(* PLC project Semester-Project-RLW, Unknown RLW-PLC-Command 0.0.1 *)
(* stored: creationDateTime 2024-10-23T22:26:44, modificationDateTime 2024-11-23T23:37:16, version 0.0.1 *)

FUNCTION isWithin5Percent : BOOL
  VAR_INPUT
    In0 : INT;
    In1 : INT;
  END_VAR
  VAR
    RangeHigh : INT;
    RangeLow : INT;
    In0IsLessThanHigh : BOOL;
    In0IsGreaterThanLow : BOOL;
  END_VAR

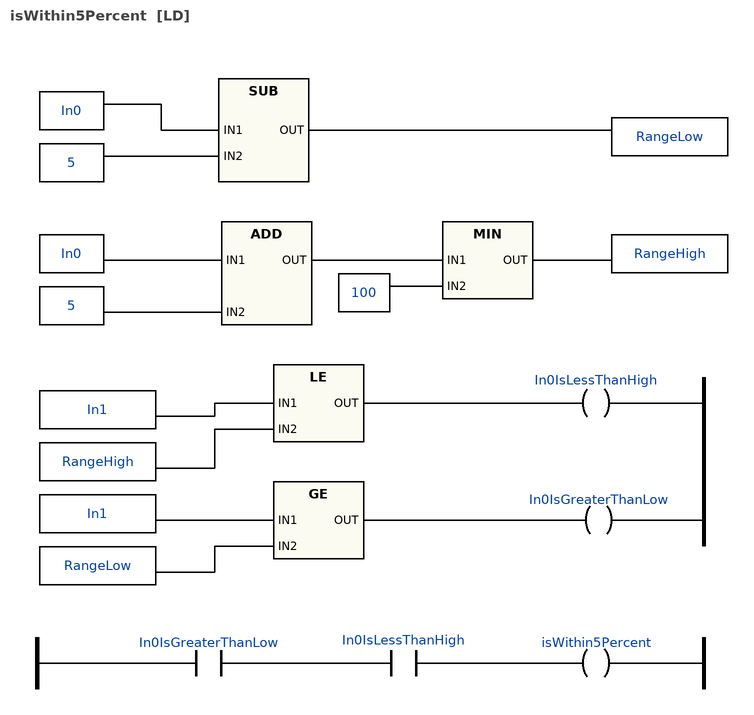
(* LD diagram, written out as Structured Text *)
RangeLow := In0 - 5;
RangeHigh := MIN(In0 + 5, 100);
In0IsLessThanHigh := In1 <= RangeHigh;
In0IsGreaterThanLow := In1 >= RangeLow;
isWithin5Percent := In0IsGreaterThanLow AND In0IsLessThanHigh;
END_FUNCTION

(* Based upon boolean inputs, returns a precentage that the isolation valve should close at. *)
FUNCTION SelectIsolationValveValue : INT
  VAR_INPUT
    SiteAlarmOverride : BOOL;  (* If high, override real num output to 0.0 *)
    BoosterPumpLogicalStatus : BOOL;  (* If high, means booster pump is working and isolation valve output should be 1.0, if low, default to 0.5 *)
  END_VAR

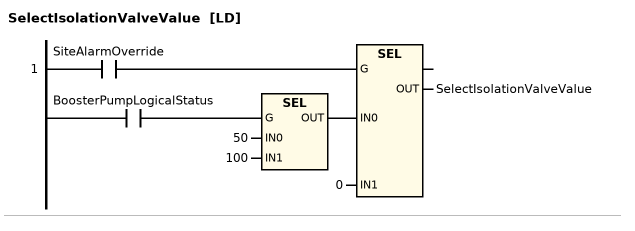
(* LD diagram, written out as Structured Text *)
SelectIsolationValveValue := SEL(SiteAlarmOverride, SEL(BoosterPumpLogicalStatus, 50, 100), 0);
END_FUNCTION

FUNCTION SetFlowSensorAlarm : BOOL
  VAR_INPUT
    IsolationValveStatus : INT;
    FlowRateSensor : INT;
  END_VAR

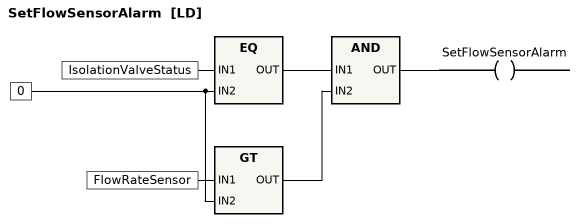
(* LD diagram, written out as Structured Text *)
SetFlowSensorAlarm := IsolationValveStatus = 0 AND FlowRateSensor > 0;
END_FUNCTION

PROGRAM DCSProgramSector
  VAR
    FlowRateSensor0 AT %IW0 : INT := 20;
    FlowRateSensor1 AT %IW1 : INT := 33;
    FlowRateSensor2 AT %IW2 : INT := 46;
    BoosterPumpStatus0 AT %IX0.0 : BOOL := True;
    BoosterPumpStatus1 AT %IX0.1 : BOOL := False;
    BoosterPumpStatus2 AT %IX0.2 : BOOL := False;
    IsolationValveStatus0 AT %IW3 : INT := 50;
    IsolationValveStatus1 AT %IW4 : INT := 50;
    IsolationValveStatus2 AT %IW5 : INT := 50;
    GeneralSiteAlarm0 AT %IX0.3 : BOOL := False;
  END_VAR
  VAR_EXTERNAL
    BoosterPumpCommand0 : BOOL;
    BoosterPumpCommand1 : BOOL;
    BoosterPumpCommand2 : BOOL;
  END_VAR
  VAR
    BoosterPumpAlarm0 AT %QX0.5 : BOOL;
    BoosterPumpAlarm1 AT %QX0.6 : BOOL;
    BoosterPumpAlarm2 AT %QX0.7 : BOOL;
    IsolationValveAlarm0 AT %QX1.0 : BOOL;
    IsolationValveAlarm1 AT %QX1.1 : BOOL;
    IsolationValveAlarm2 AT %QX1.2 : BOOL;
    FlowSensorAlarm0 AT %QX1.3 : BOOL;
    FlowSensorAlarm1 AT %QX1.4 : BOOL;
    FlowSensorAlarm2 AT %QX1.5 : BOOL;
    FlowRateAlarm0 AT %QX4.3 : BOOL;
    FlowRateAlarm1 AT %QX4.4 : BOOL;
    FlowRateAlarm2 AT %QX4.5 : BOOL;
  END_VAR
  VAR_EXTERNAL
    IsolationValveCommand0 : INT;
    IsolationValveCommand1 : INT;
    IsolationValveCommand2 : INT;
  END_VAR
  VAR CONSTANT
    FlowSensorMaxCapacity AT %MW0 : INT := 50;
  END_VAR
  VAR  (* added by the conversion: wires and edge detectors of the diagram *)
    _SelectIsolationValveValue19_OUT : INT;
    _SelectIsolationValveValue25_OUT : INT;
    _SelectIsolationValveValue92_OUT : INT;
  END_VAR

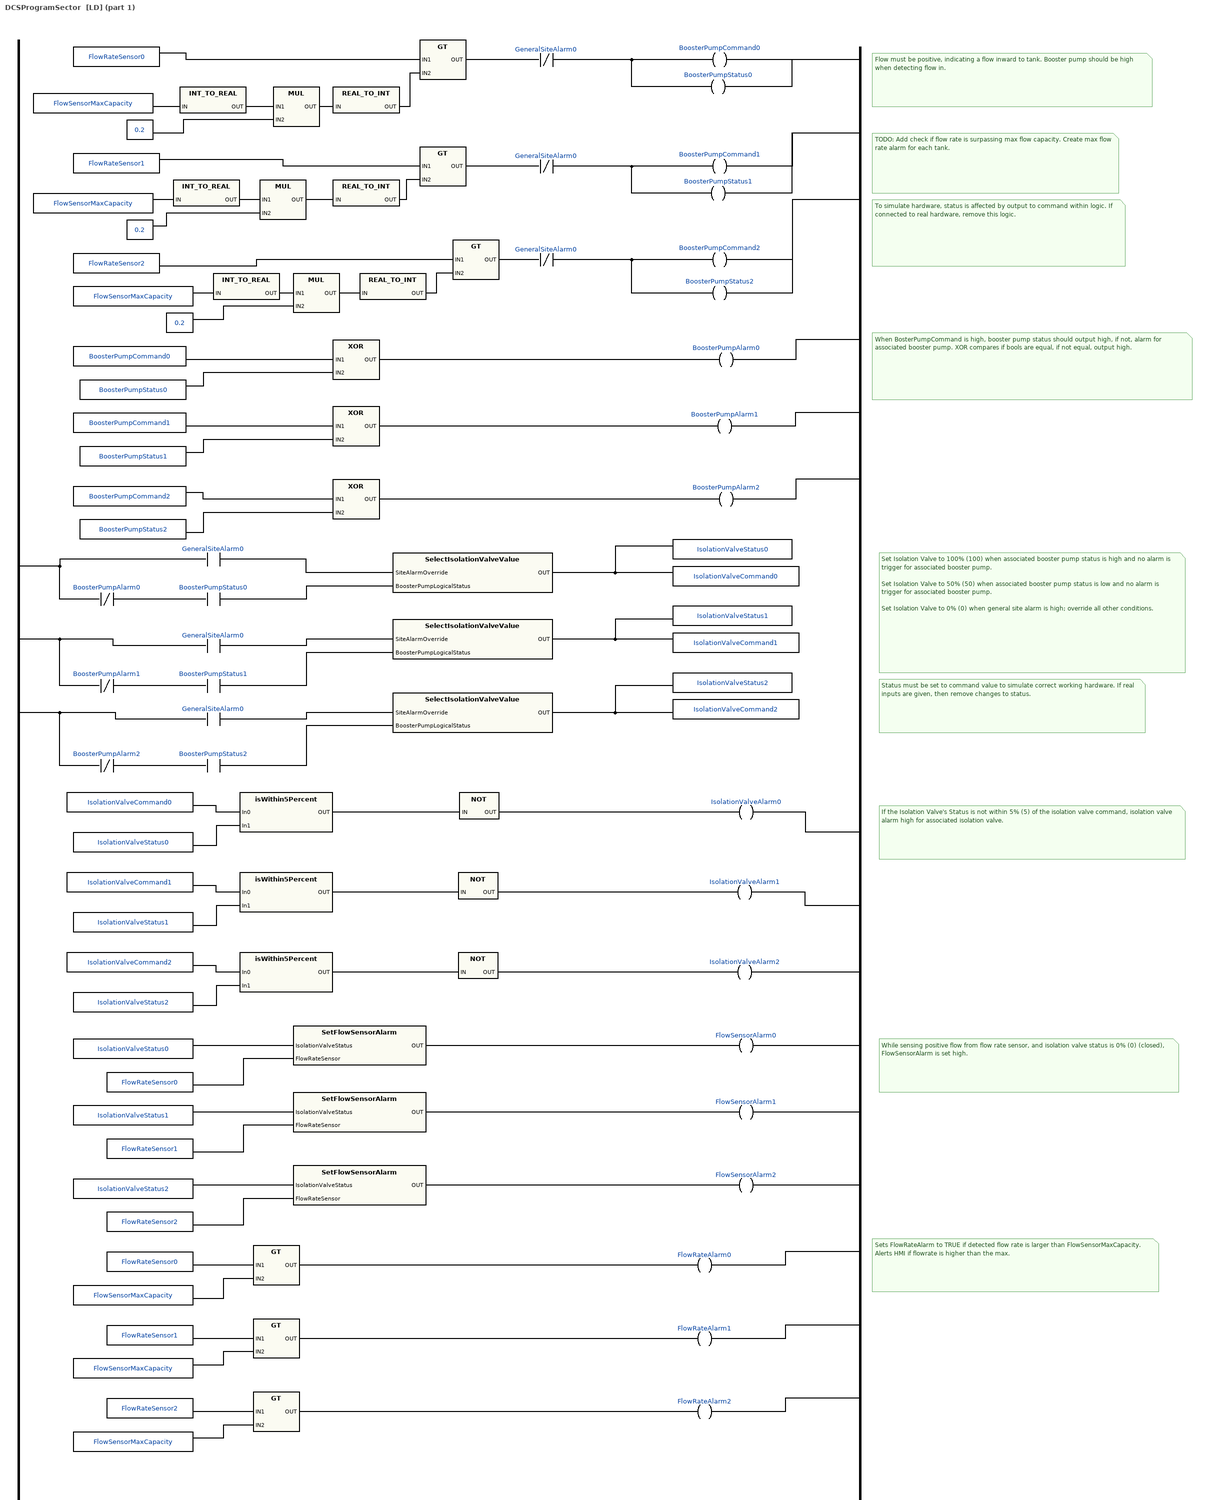
(* LD diagram, written out as Structured Text *)
(* Flow must be positive, indicating a flow inward to tank. Booster pump should be high when detecting flow in. *)
BoosterPumpCommand0 := FlowRateSensor0 > REAL_TO_INT(INT_TO_REAL(FlowSensorMaxCapacity) * 0.2) AND NOT GeneralSiteAlarm0;
(* TODO: Add check if flow rate is surpassing max flow capacity. Create max flow rate alarm for each tank. *)
BoosterPumpCommand1 := FlowRateSensor1 > REAL_TO_INT(INT_TO_REAL(FlowSensorMaxCapacity) * 0.2) AND NOT GeneralSiteAlarm0;
(* To simulate hardware, status is affected by output to command within logic. If connected to real hardware, remove this logic. *)
BoosterPumpCommand2 := FlowRateSensor2 > REAL_TO_INT(INT_TO_REAL(FlowSensorMaxCapacity) * 0.2) AND NOT GeneralSiteAlarm0;
(* When BosterPumpCommand is high, booster pump status should output high, if not, alarm for associated booster pump. XOR compares if bools are equal, if not equal, output high. *)
BoosterPumpAlarm0 := BoosterPumpCommand0 XOR BoosterPumpStatus0;
BoosterPumpAlarm2 := BoosterPumpCommand2 XOR BoosterPumpStatus2;
(* Set Isolation Valve to 100% (100) when associated booster pump status is high and no alarm is trigger for associated booster pump.

Set Isolation Valve to 50% (50) when associated booster pump status is low and no alarm is trigger for associated booster pump.

Set Isolation Valve to 0% (0) when general site alarm is high; override all other conditions. *)
_SelectIsolationValveValue19_OUT := SelectIsolationValveValue(GeneralSiteAlarm0, NOT BoosterPumpAlarm1 AND BoosterPumpStatus1);
IsolationValveCommand1 := _SelectIsolationValveValue19_OUT;
(* Status must be set to command value to simulate correct working hardware. If real inputs are given, then remove changes to status. *)
_SelectIsolationValveValue25_OUT := SelectIsolationValveValue(GeneralSiteAlarm0, NOT BoosterPumpAlarm2 AND BoosterPumpStatus2);
IsolationValveCommand2 := _SelectIsolationValveValue25_OUT;
(* If the Isolation Valve's Status is not within 5% (5) of the isolation valve command, isolation valve alarm high for associated isolation valve. *)
IsolationValveAlarm0 := NOT isWithin5Percent(IsolationValveCommand0, IsolationValveStatus0);
IsolationValveAlarm1 := NOT isWithin5Percent(IsolationValveCommand1, IsolationValveStatus1);
IsolationValveAlarm2 := NOT isWithin5Percent(IsolationValveCommand2, IsolationValveStatus2);
BoosterPumpAlarm1 := BoosterPumpCommand1 XOR BoosterPumpStatus1;
_SelectIsolationValveValue92_OUT := SelectIsolationValveValue(GeneralSiteAlarm0, NOT BoosterPumpAlarm0 AND BoosterPumpStatus0);
IsolationValveCommand0 := _SelectIsolationValveValue92_OUT;
(* While sensing positive flow from flow rate sensor, and isolation valve status is 0% (0) (closed), FlowSensorAlarm is set high. *)
FlowSensorAlarm0 := SetFlowSensorAlarm(IsolationValveStatus0, FlowRateSensor0);
FlowSensorAlarm1 := SetFlowSensorAlarm(IsolationValveStatus1, FlowRateSensor1);
FlowSensorAlarm2 := SetFlowSensorAlarm(IsolationValveStatus2, FlowRateSensor2);
IsolationValveStatus0 := _SelectIsolationValveValue92_OUT;
IsolationValveStatus1 := _SelectIsolationValveValue19_OUT;
IsolationValveStatus2 := _SelectIsolationValveValue25_OUT;
BoosterPumpStatus0 := FlowRateSensor0 > REAL_TO_INT(INT_TO_REAL(FlowSensorMaxCapacity) * 0.2) AND NOT GeneralSiteAlarm0;
BoosterPumpStatus1 := FlowRateSensor1 > REAL_TO_INT(INT_TO_REAL(FlowSensorMaxCapacity) * 0.2) AND NOT GeneralSiteAlarm0;
BoosterPumpStatus2 := FlowRateSensor2 > REAL_TO_INT(INT_TO_REAL(FlowSensorMaxCapacity) * 0.2) AND NOT GeneralSiteAlarm0;
(* Sets FlowRateAlarm to TRUE if detected flow rate is larger than FlowSensorMaxCapacity. Alerts HMI if flowrate is higher than the max. *)
FlowRateAlarm0 := FlowRateSensor0 > FlowSensorMaxCapacity;
FlowRateAlarm1 := FlowRateSensor1 > FlowSensorMaxCapacity;
FlowRateAlarm2 := FlowRateSensor2 > FlowSensorMaxCapacity;
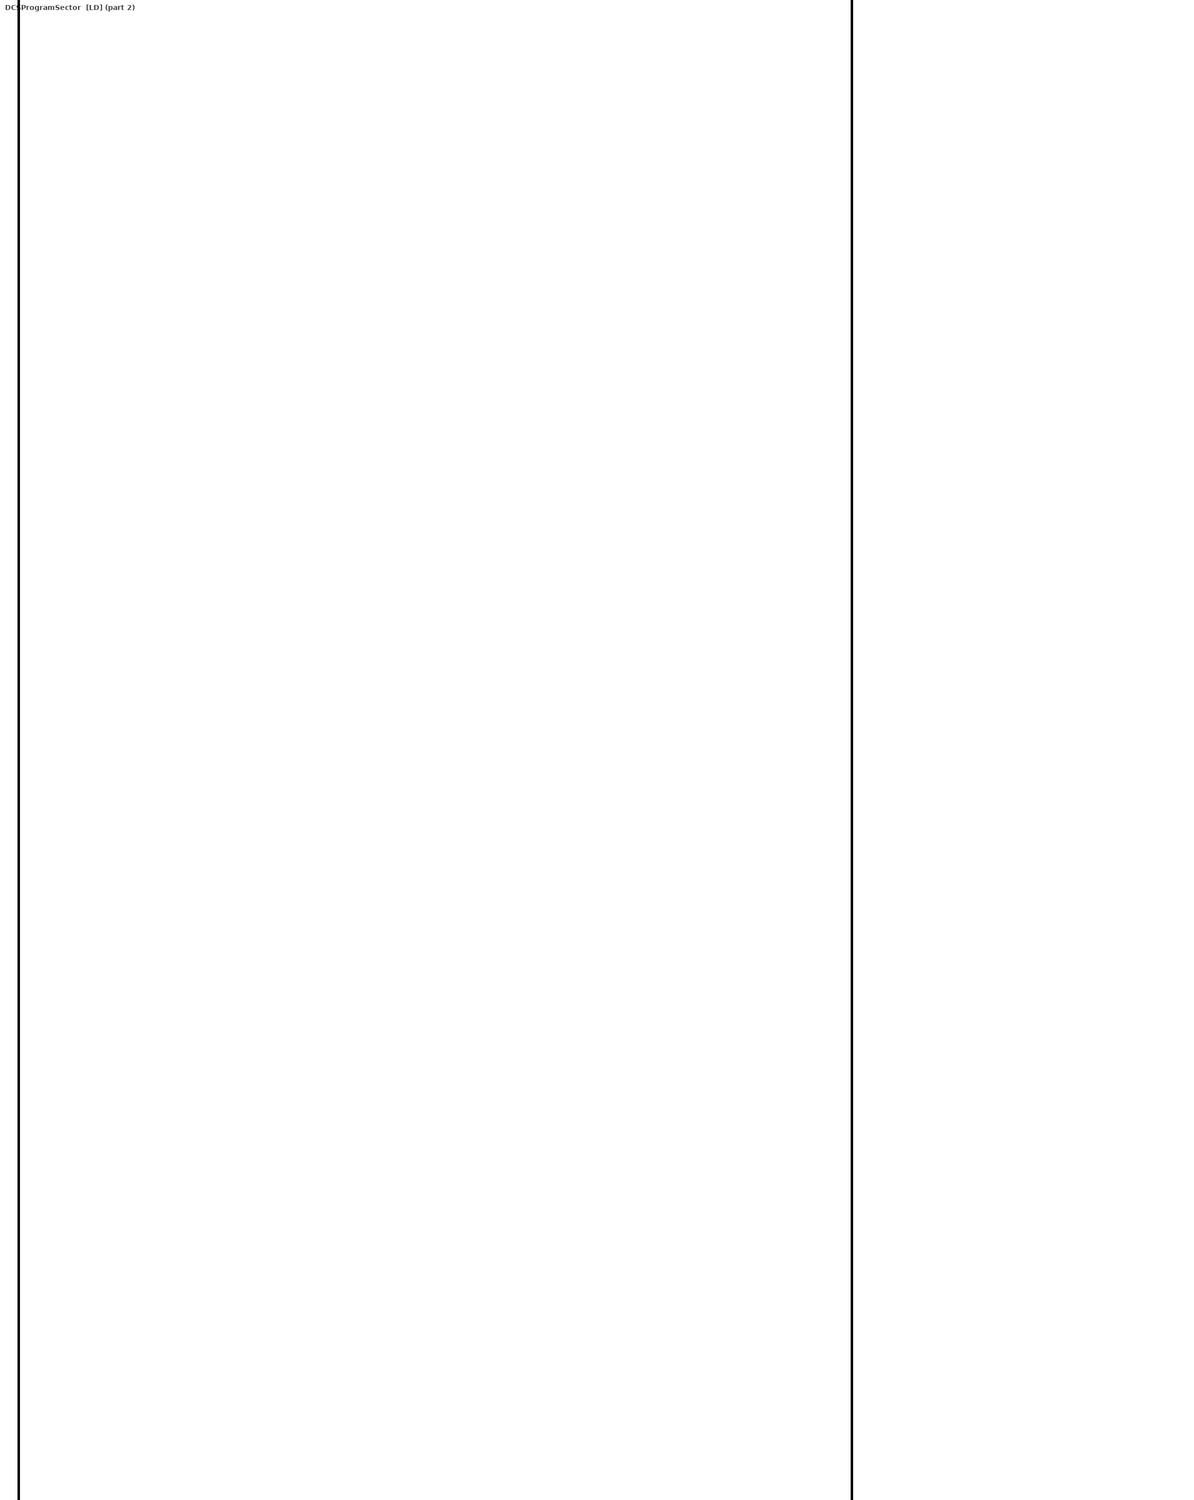
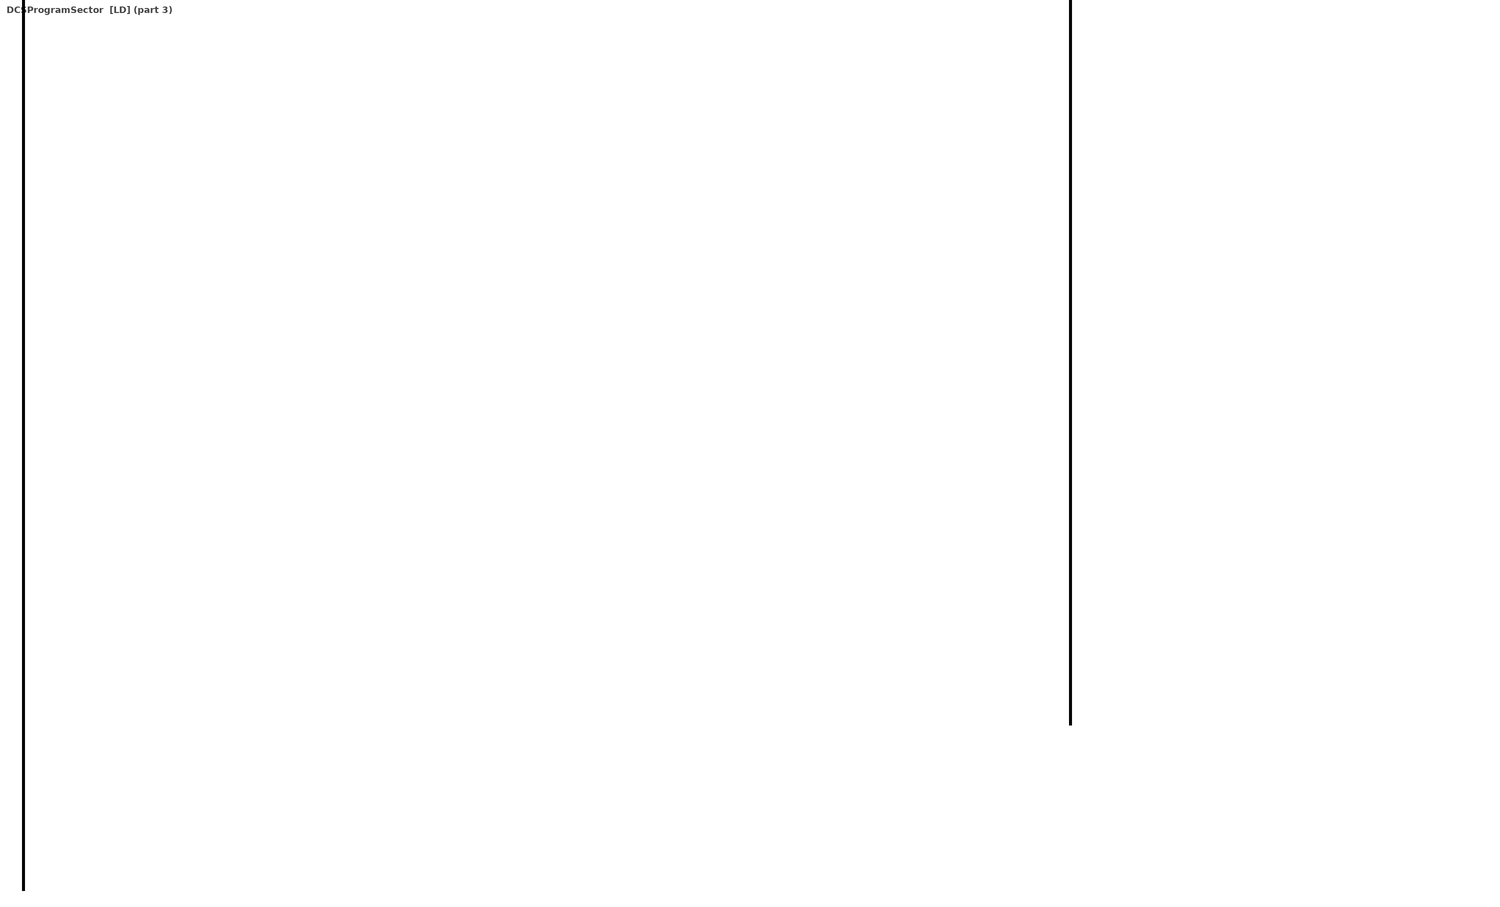
END_PROGRAM

FUNCTION_BLOCK DisposalProtocol
  VAR_INPUT
    In : BOOL;
    DistributionPumpSpeedIn : INT;
    DisposalValveCommandIn : INT;
  END_VAR
  VAR_OUTPUT
    Out : BOOL;
    DistributionPumpSpeedOut : INT;
    DisposalValveCommandOut : INT;
  END_VAR
  VAR  (* added by the conversion: wires and edge detectors of the diagram *)
    _MOVE3_ENO : BOOL;
    _MOVE3_OUT : INT;
    _MOVE6_ENO : BOOL;
    _MOVE6_OUT : INT;
  END_VAR

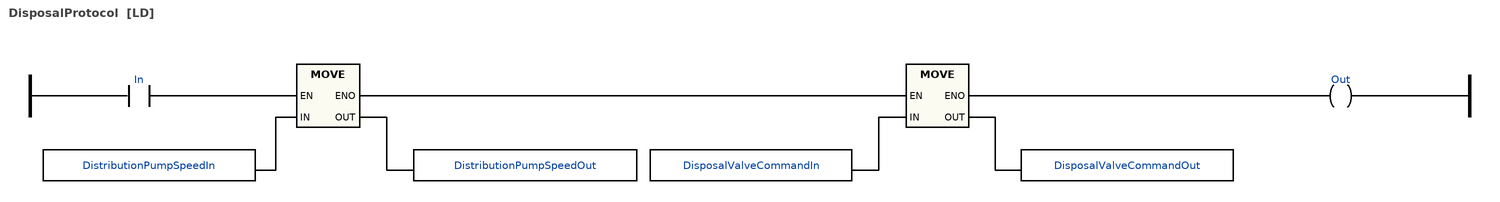
(* LD diagram, written out as Structured Text *)
_MOVE3_OUT := MOVE(EN := In, IN := DistributionPumpSpeedIn, ENO => _MOVE3_ENO);
IF _MOVE3_ENO THEN DistributionPumpSpeedOut := _MOVE3_OUT; END_IF;
_MOVE6_OUT := MOVE(EN := _MOVE3_ENO, IN := DisposalValveCommandIn, ENO => _MOVE6_ENO);
IF _MOVE6_ENO THEN DisposalValveCommandOut := _MOVE6_OUT; END_IF;
Out := _MOVE6_ENO;
END_FUNCTION_BLOCK

(* Set the distribution pump speed based upon the number of open eductor valves and if there is detected high pressure in one of the tanks. *)
FUNCTION SetDistributionPumpSpeed : INT
  VAR_INPUT
    isEductorValve0Open : BOOL;
    isEductorValve1Open : BOOL;
    isEductorValve2Open : BOOL;
    isDistributionPumpSpeedReduction : BOOL;
  END_VAR
  VAR  (* added by the conversion: wires and edge detectors of the diagram *)
    _MOVE7_ENO : BOOL;
    _MOVE7_OUT : INT;
    _MOVE8_ENO : BOOL;
    _MOVE8_OUT : INT;
    _MOVE9_ENO : BOOL;
    _MOVE9_OUT : INT;
    _MOVE10_ENO : BOOL;
    _MOVE10_OUT : INT;
  END_VAR

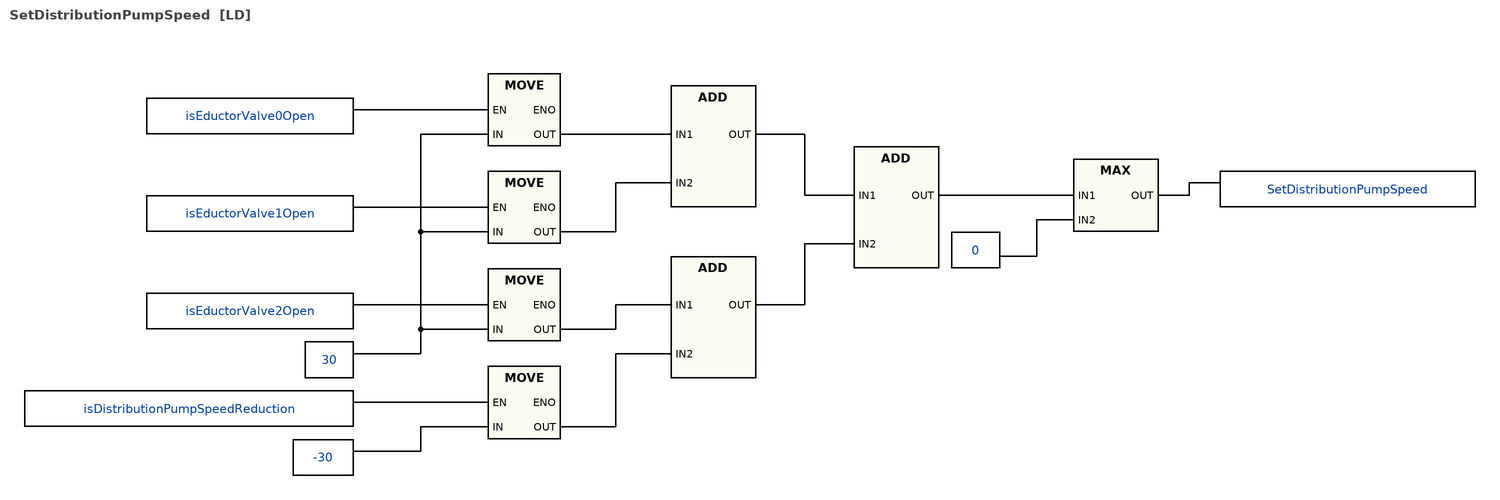
(* LD diagram, written out as Structured Text *)
_MOVE7_OUT := MOVE(EN := isEductorValve0Open, IN := 30, ENO => _MOVE7_ENO);
_MOVE8_OUT := MOVE(EN := isEductorValve1Open, IN := 30, ENO => _MOVE8_ENO);
_MOVE9_OUT := MOVE(EN := isEductorValve2Open, IN := 30, ENO => _MOVE9_ENO);
_MOVE10_OUT := MOVE(EN := isDistributionPumpSpeedReduction, IN := -30, ENO => _MOVE10_ENO);
SetDistributionPumpSpeed := MAX(_MOVE7_OUT + _MOVE8_OUT + (_MOVE9_OUT + _MOVE10_OUT), 0);
END_FUNCTION

(* Given a pulse in, output a true boolean to DistributionPumpOut and 0.0 to EductorValveOut *)
FUNCTION_BLOCK Tank15MinuteReset
  VAR_INPUT
    PulseIn : BOOL;
  END_VAR
  VAR_OUTPUT
    DistributionPumpOut : BOOL;
    EductorValveOut : INT;
  END_VAR
  VAR
    TON1 : TON;
    TP1 : TP;
  END_VAR
  VAR  (* added by the conversion: wires and edge detectors of the diagram *)
    _MOVE100_ENO : BOOL;
    _MOVE100_OUT : INT;
  END_VAR

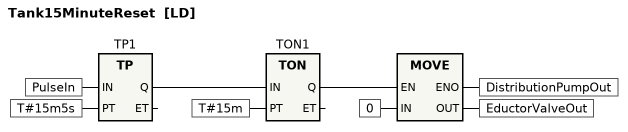
(* LD diagram, written out as Structured Text *)
TP1(IN := PulseIn, PT := T#15m5s);
TON1(IN := TP1.Q, PT := T#15m);
_MOVE100_OUT := MOVE(EN := TON1.Q, IN := 0, ENO => _MOVE100_ENO);
DistributionPumpOut := _MOVE100_ENO;
IF _MOVE100_ENO THEN EductorValveOut := _MOVE100_OUT; END_IF;
END_FUNCTION_BLOCK

PROGRAM SCADATankLevelProgram
  VAR
    EductorValveStatus0 AT %IW6 : INT;
    EductorValveStatus1 AT %IW7 : INT;
    EductorValveStatus2 AT %IW8 : INT;
    UltrasonicTankLevelSensor0 AT %IW9 : INT := 20;
    UltrasonicTankLevelSensor1 AT %IW10 : INT := 15;
    UltrasonicTankLevelSensor2 AT %IW11 : INT := 17;
    DisposalValveStatus AT %IW12 : INT := 0;
    DistributionPumpStatus AT %IX0.4 : BOOL;
    HighPressureSwitch0 AT %IX0.5 : BOOL;
    HighPressureSwitch1 AT %IX0.6 : BOOL;
    HighPressureSwitch2 AT %IX0.7 : BOOL;
    EductorValveCommand0 AT %QW3 : INT := 0;
    EductorValveCommand1 AT %QW4 : INT := 0;
    EductorValveCommand2 AT %QW5 : INT := 0;
    EductorValveAlarm0 AT %QX1.6 : BOOL;
    EductorValveAlarm1 AT %QX1.7 : BOOL;
    EductorValveAlarm2 AT %QX2.0 : BOOL;
    DistributionPumpCommand AT %QX2.1 : BOOL;
    DistributionPumpSpeedCommand AT %QW6 : INT := 0;
    DisposalValveCommand AT %QW7 : INT := 0;
    DistributionPumpPressureReductionFlag AT %MX0.2 : BOOL;
    Tank30Capacity0 AT %MX0.3 : BOOL;
    Tank30Capacity1 AT %MX0.4 : BOOL;
    Tank30Capacity2 AT %MX0.5 : BOOL;
    Tank60Capacity0 AT %MX0.6 : BOOL;
    Tank60Capacity1 AT %MX0.7 : BOOL;
    Tank60Capacity2 AT %MX1.0 : BOOL;
    Tank90Capacity0 AT %MX1.2 : BOOL;
    Tank90Capacity1 AT %MX1.3 : BOOL;
    Tank90Capacity2 AT %MX1.4 : BOOL;
    isTank0DisposalReady AT %MX1.5 : BOOL;
    isTank1DisposalReady AT %MX1.6 : BOOL;
    isTank2DisposalReady AT %MX1.7 : BOOL;
    AllTanksNearCapacity AT %MX2.0 : BOOL;
    DistributionPumpAlarm AT %QX2.2 : BOOL;
    HighPressureSwitchAlarm0 AT %QX2.3 : BOOL;
    HighPressureSwitchAlarm1 AT %QX2.4 : BOOL;
    HighPressureSwitchAlarm2 AT %QX2.5 : BOOL;
    askHMIContainmentUnitAttached AT %QX2.6 : BOOL;
    askHMIContainmentUnitFull AT %QX2.7 : BOOL;
    DisposalValveAlarm AT %QX3.0 : BOOL;
    TankCapacityAlarm0 AT %QX3.1 : BOOL;
    TankCapacityAlarm1 AT %QX3.2 : BOOL;
    TankCapacityAlarm2 AT %QX3.3 : BOOL;
    CentralTankAlarmSwitch AT %QX3.4 : BOOL;
    ControlCenterHornStrobeAlarm AT %QX3.5 : BOOL;
    pHWarningHMI AT %QX3.6 : BOOL;
    pHCriticalHMI AT %QX3.7 : BOOL;
    HMITankDisposalButton AT %QX4.0 : BOOL;
    isContainmentUnitAttached AT %QX4.1 : BOOL;
    isContainmentUnitFull AT %QX4.2 : BOOL;
  END_VAR
  VAR_EXTERNAL
    BoosterPumpCommand0 : BOOL;  (* External Global Variable Utilized by the DCS Program *)
    BoosterPumpCommand1 : BOOL;
    BoosterPumpCommand2 : BOOL;
    IsolationValveCommand0 : INT;
    IsolationValveCommand1 : INT;
    IsolationValveCommand2 : INT;
    pHAlertAlarm : BOOL;
    pHCriticalAlarm : BOOL;
  END_VAR
  VAR
    Tank15MinuteReset0 : Tank15MinuteReset;
    Tank15MinuteReset1 : Tank15MinuteReset;
    Tank15MinuteReset2 : Tank15MinuteReset;
    DisposalProtocol0 : DisposalProtocol;
    DisposalProtocol1 : DisposalProtocol;
  END_VAR
  VAR  (* added by the conversion: wires and edge detectors of the diagram *)
    R_TRIG1 : R_TRIG;
    _MOVE84_ENO : BOOL;
    _MOVE84_OUT : INT;
    R_TRIG2 : R_TRIG;
    _MOVE89_ENO : BOOL;
    _MOVE89_OUT : INT;
    R_TRIG3 : R_TRIG;
    _MOVE94_ENO : BOOL;
    _MOVE94_OUT : INT;
    R_TRIG4 : R_TRIG;
    R_TRIG5 : R_TRIG;
    R_TRIG6 : R_TRIG;
    _MOVE146_ENO : BOOL;
    _MOVE146_OUT : INT;
    _MOVE117_ENO : BOOL;
    _MOVE117_OUT : INT;
    _MOVE132_ENO : BOOL;
    _MOVE132_OUT : INT;
    _MOVE200_ENO : BOOL;
    _MOVE200_OUT : INT;
    _MOVE111_ENO : BOOL;
    _MOVE111_OUT : INT;
    _MOVE143_ENO : BOOL;
    _MOVE143_OUT : INT;
    _MOVE156_ENO : BOOL;
    _MOVE156_OUT : INT;
  END_VAR

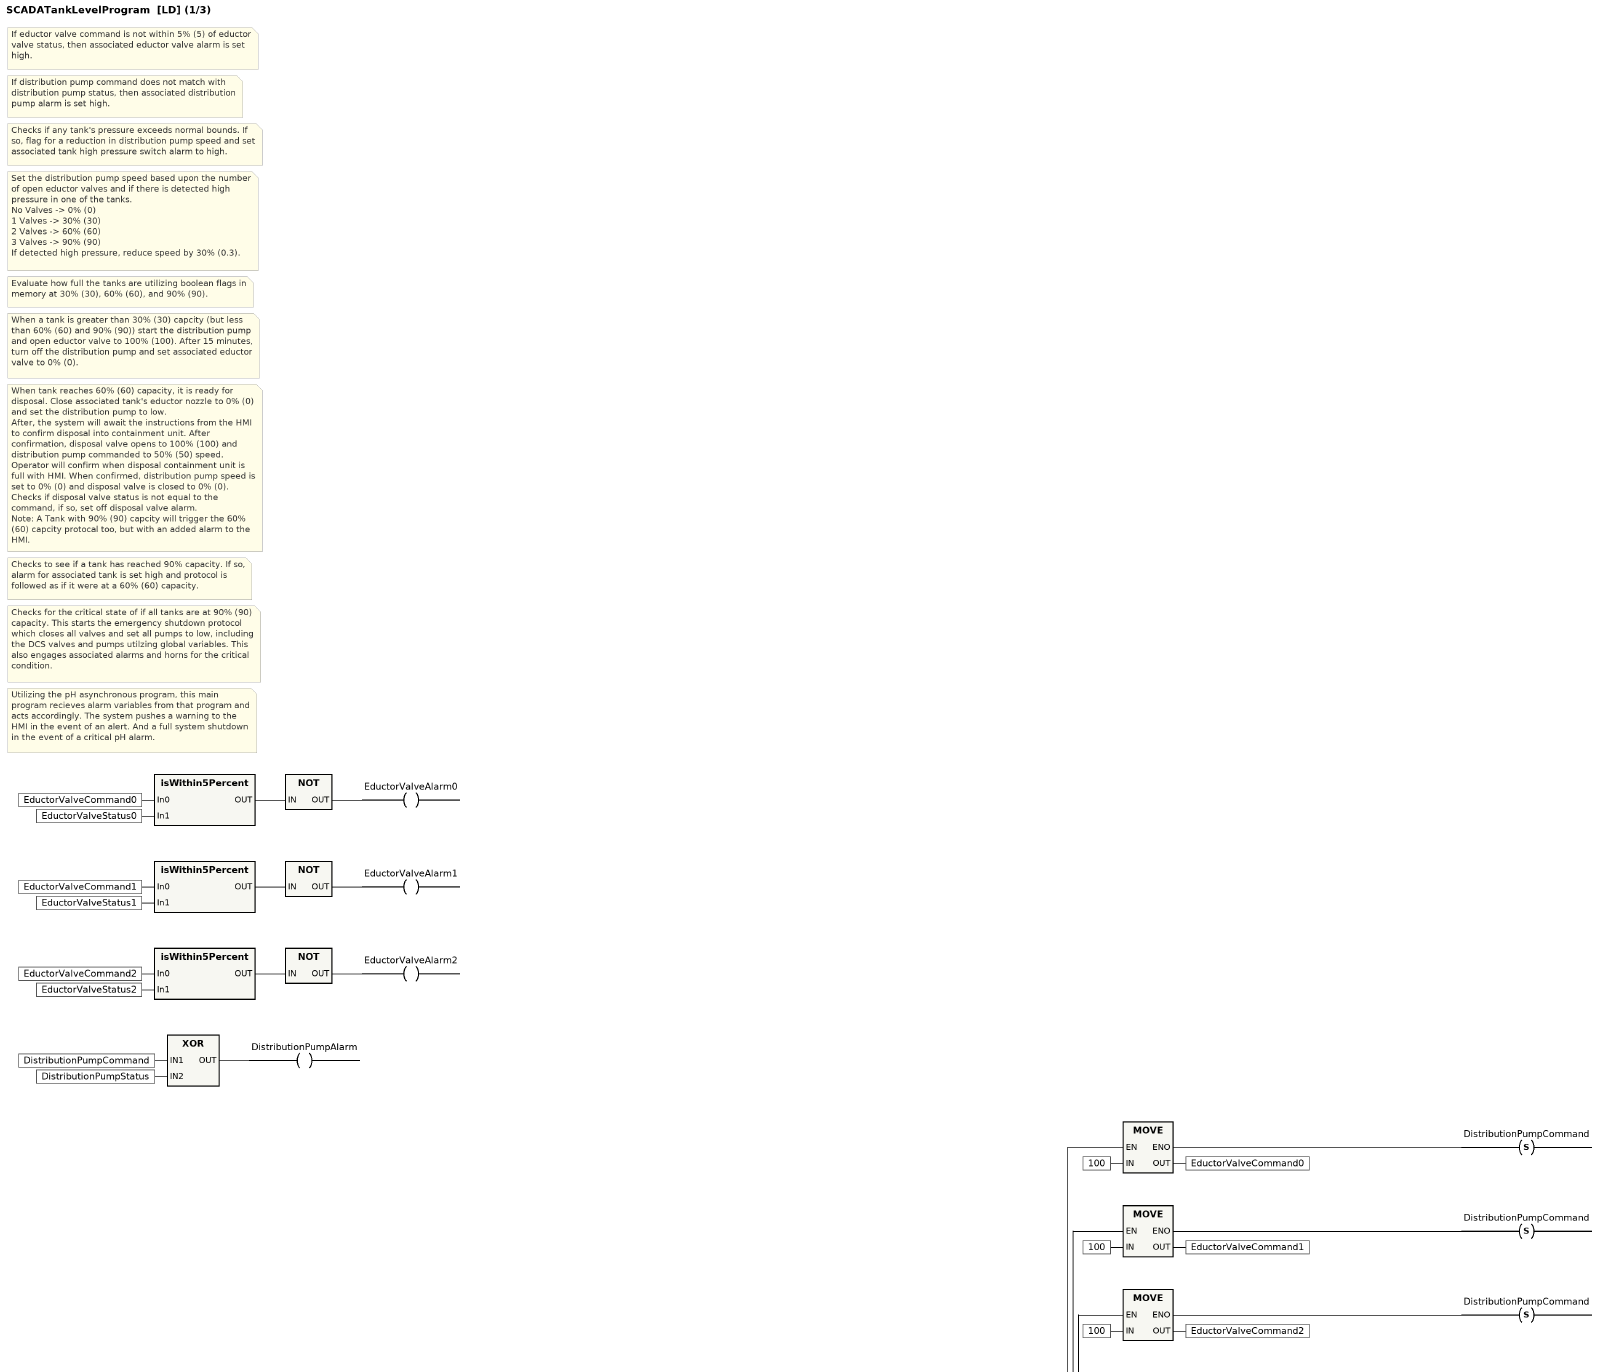
(* LD diagram, written out as Structured Text *)
(* If eductor valve command is not within 5% (5) of eductor valve status, then associated eductor valve alarm is set high. *)
EductorValveAlarm0 := NOT isWithin5Percent(EductorValveCommand0, EductorValveStatus0);
EductorValveAlarm1 := NOT isWithin5Percent(EductorValveCommand1, EductorValveStatus1);
EductorValveAlarm2 := NOT isWithin5Percent(EductorValveCommand2, EductorValveStatus2);
(* If distribution pump command does not match with distribution pump status, then associated distribution pump alarm is set high. *)
DistributionPumpAlarm := DistributionPumpCommand XOR DistributionPumpStatus;
(* Checks if any tank's pressure exceeds normal bounds. If so, flag for a reduction in distribution pump speed and set associated tank high pressure switch alarm to high. *)
HighPressureSwitchAlarm0 := HighPressureSwitch0;
HighPressureSwitchAlarm1 := HighPressureSwitch1;
HighPressureSwitchAlarm2 := HighPressureSwitch2;
DistributionPumpPressureReductionFlag := HighPressureSwitch0 OR HighPressureSwitch1 OR HighPressureSwitch2;
DistributionPumpSpeedCommand := SetDistributionPumpSpeed(isWithin5Percent(EductorValveStatus0, 100), isWithin5Percent(EductorValveStatus1, 100), isWithin5Percent(EductorValveStatus2, 100), DistributionPumpPressureReductionFlag);
(* Set the distribution pump speed based upon the number of open eductor valves and if there is detected high pressure in one of the tanks.
No Valves -> 0% (0)
1 Valves -> 30% (30)
2 Valves -> 60% (60)
3 Valves -> 90% (90)
If detected high pressure, reduce speed by 30% (0.3). *)
(* Evaluate how full the tanks are utilizing boolean flags in memory at 30% (30), 60% (60), and 90% (90). *)
Tank30Capacity0 := UltrasonicTankLevelSensor0 >= 30;
Tank30Capacity1 := UltrasonicTankLevelSensor1 >= 30;
Tank30Capacity2 := UltrasonicTankLevelSensor2 >= 30;
Tank60Capacity0 := UltrasonicTankLevelSensor0 >= 60;
Tank60Capacity1 := UltrasonicTankLevelSensor1 >= 60;
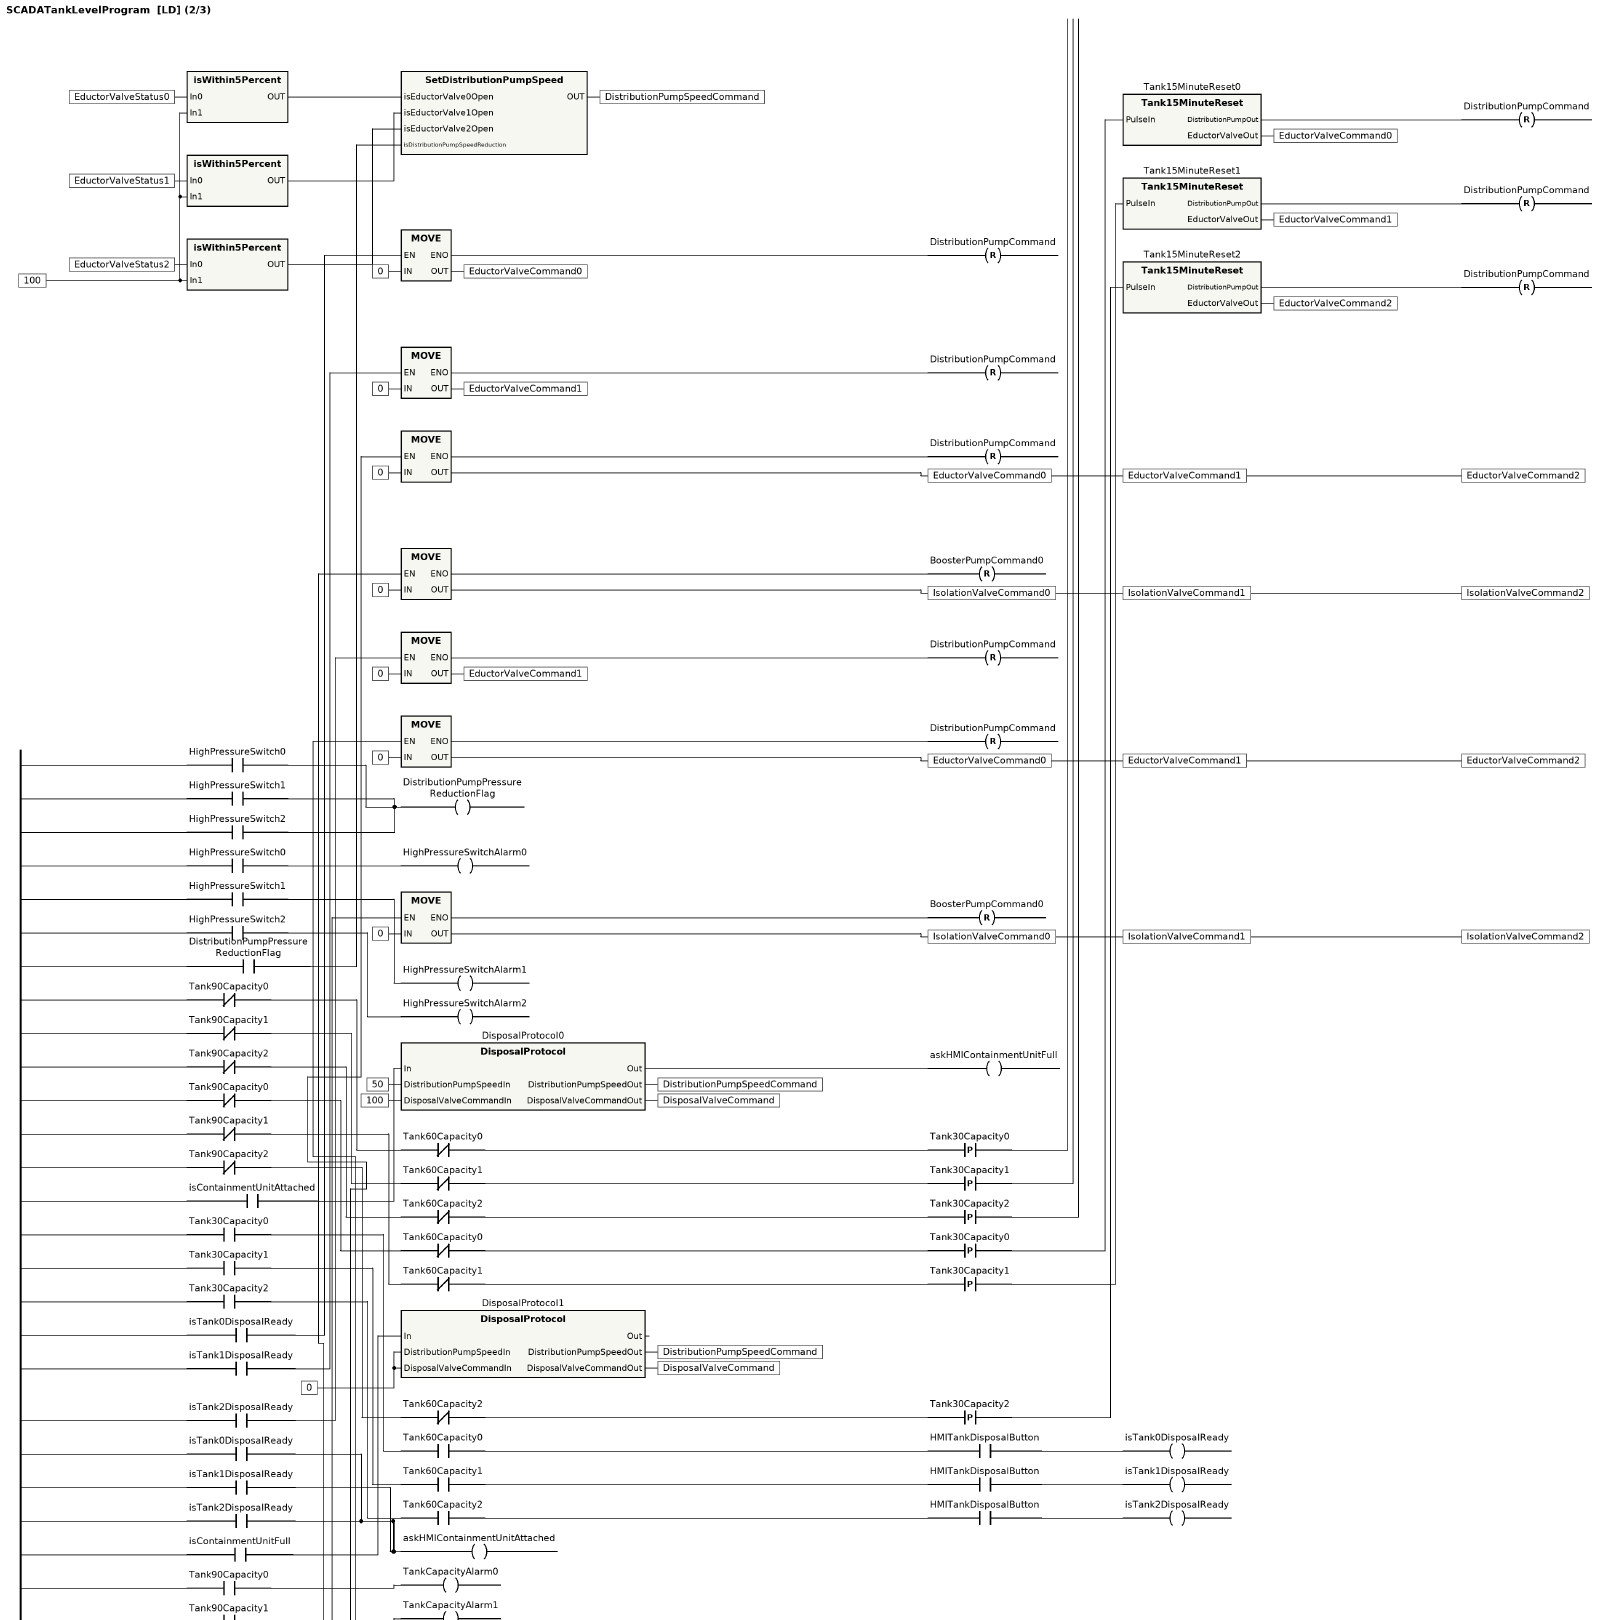
Tank60Capacity2 := UltrasonicTankLevelSensor2 >= 60;
Tank90Capacity0 := UltrasonicTankLevelSensor0 >= 90;
Tank90Capacity1 := UltrasonicTankLevelSensor1 >= 90;
Tank90Capacity2 := UltrasonicTankLevelSensor2 >= 90;
(* When a tank is greater than 30% (30) capcity (but less than 60% (60) and 90% (90)) start the distribution pump and open eductor valve to 100% (100). After 15 minutes, turn off the distribution pump and set associated eductor valve to 0% (0). *)
R_TRIG1(CLK := Tank30Capacity0);
_MOVE84_OUT := MOVE(EN := NOT Tank90Capacity0 AND NOT Tank60Capacity0 AND R_TRIG1.Q, IN := 100, ENO => _MOVE84_ENO);
IF _MOVE84_ENO THEN EductorValveCommand0 := _MOVE84_OUT; END_IF;
IF _MOVE84_ENO THEN DistributionPumpCommand := TRUE; END_IF;
R_TRIG2(CLK := Tank30Capacity1);
_MOVE89_OUT := MOVE(EN := NOT Tank90Capacity1 AND NOT Tank60Capacity1 AND R_TRIG2.Q, IN := 100, ENO => _MOVE89_ENO);
IF _MOVE89_ENO THEN DistributionPumpCommand := TRUE; END_IF;
IF _MOVE89_ENO THEN EductorValveCommand1 := _MOVE89_OUT; END_IF;
R_TRIG3(CLK := Tank30Capacity2);
_MOVE94_OUT := MOVE(EN := NOT Tank90Capacity2 AND NOT Tank60Capacity2 AND R_TRIG3.Q, IN := 100, ENO => _MOVE94_ENO);
IF _MOVE94_ENO THEN DistributionPumpCommand := TRUE; END_IF;
IF _MOVE94_ENO THEN EductorValveCommand2 := _MOVE94_OUT; END_IF;
R_TRIG4(CLK := Tank30Capacity0);
Tank15MinuteReset0(PulseIn := NOT Tank90Capacity0 AND NOT Tank60Capacity0 AND R_TRIG4.Q);
IF Tank15MinuteReset0.DistributionPumpOut THEN DistributionPumpCommand := FALSE; END_IF;
EductorValveCommand0 := Tank15MinuteReset0.EductorValveOut;
R_TRIG5(CLK := Tank30Capacity1);
Tank15MinuteReset1(PulseIn := NOT Tank90Capacity1 AND NOT Tank60Capacity1 AND R_TRIG5.Q);
EductorValveCommand1 := Tank15MinuteReset1.EductorValveOut;
IF Tank15MinuteReset1.DistributionPumpOut THEN DistributionPumpCommand := FALSE; END_IF;
R_TRIG6(CLK := Tank30Capacity2);
Tank15MinuteReset2(PulseIn := NOT Tank90Capacity2 AND NOT Tank60Capacity2 AND R_TRIG6.Q);
IF Tank15MinuteReset2.DistributionPumpOut THEN DistributionPumpCommand := FALSE; END_IF;
EductorValveCommand2 := Tank15MinuteReset2.EductorValveOut;
(* When tank reaches 60% (60) capacity, it is ready for disposal. Close associated tank's eductor nozzle to 0% (0) and set the distribution pump to low.

After, the system will await the instructions from the HMI to confirm disposal into containment unit. After confirmation, disposal valve opens to 100% (100) and distribution pump commanded to 50% (50) speed.

Operator will confirm when disposal containment unit is full with HMI. When confirmed, distribution pump speed is set to 0% (0) and disposal valve is closed to 0% (0).

Checks if disposal valve status is not equal to the command, if so, set off disposal valve alarm. 

Note: A Tank with 90% (90) capcity will trigger the 60% (60) capcity protocal too, but with an added alarm to the HMI. *)
_MOVE146_OUT := MOVE(EN := isTank0DisposalReady, IN := 0, ENO => _MOVE146_ENO);
IF _MOVE146_ENO THEN EductorValveCommand0 := _MOVE146_OUT; END_IF;
IF _MOVE146_ENO THEN DistributionPumpCommand := FALSE; END_IF;
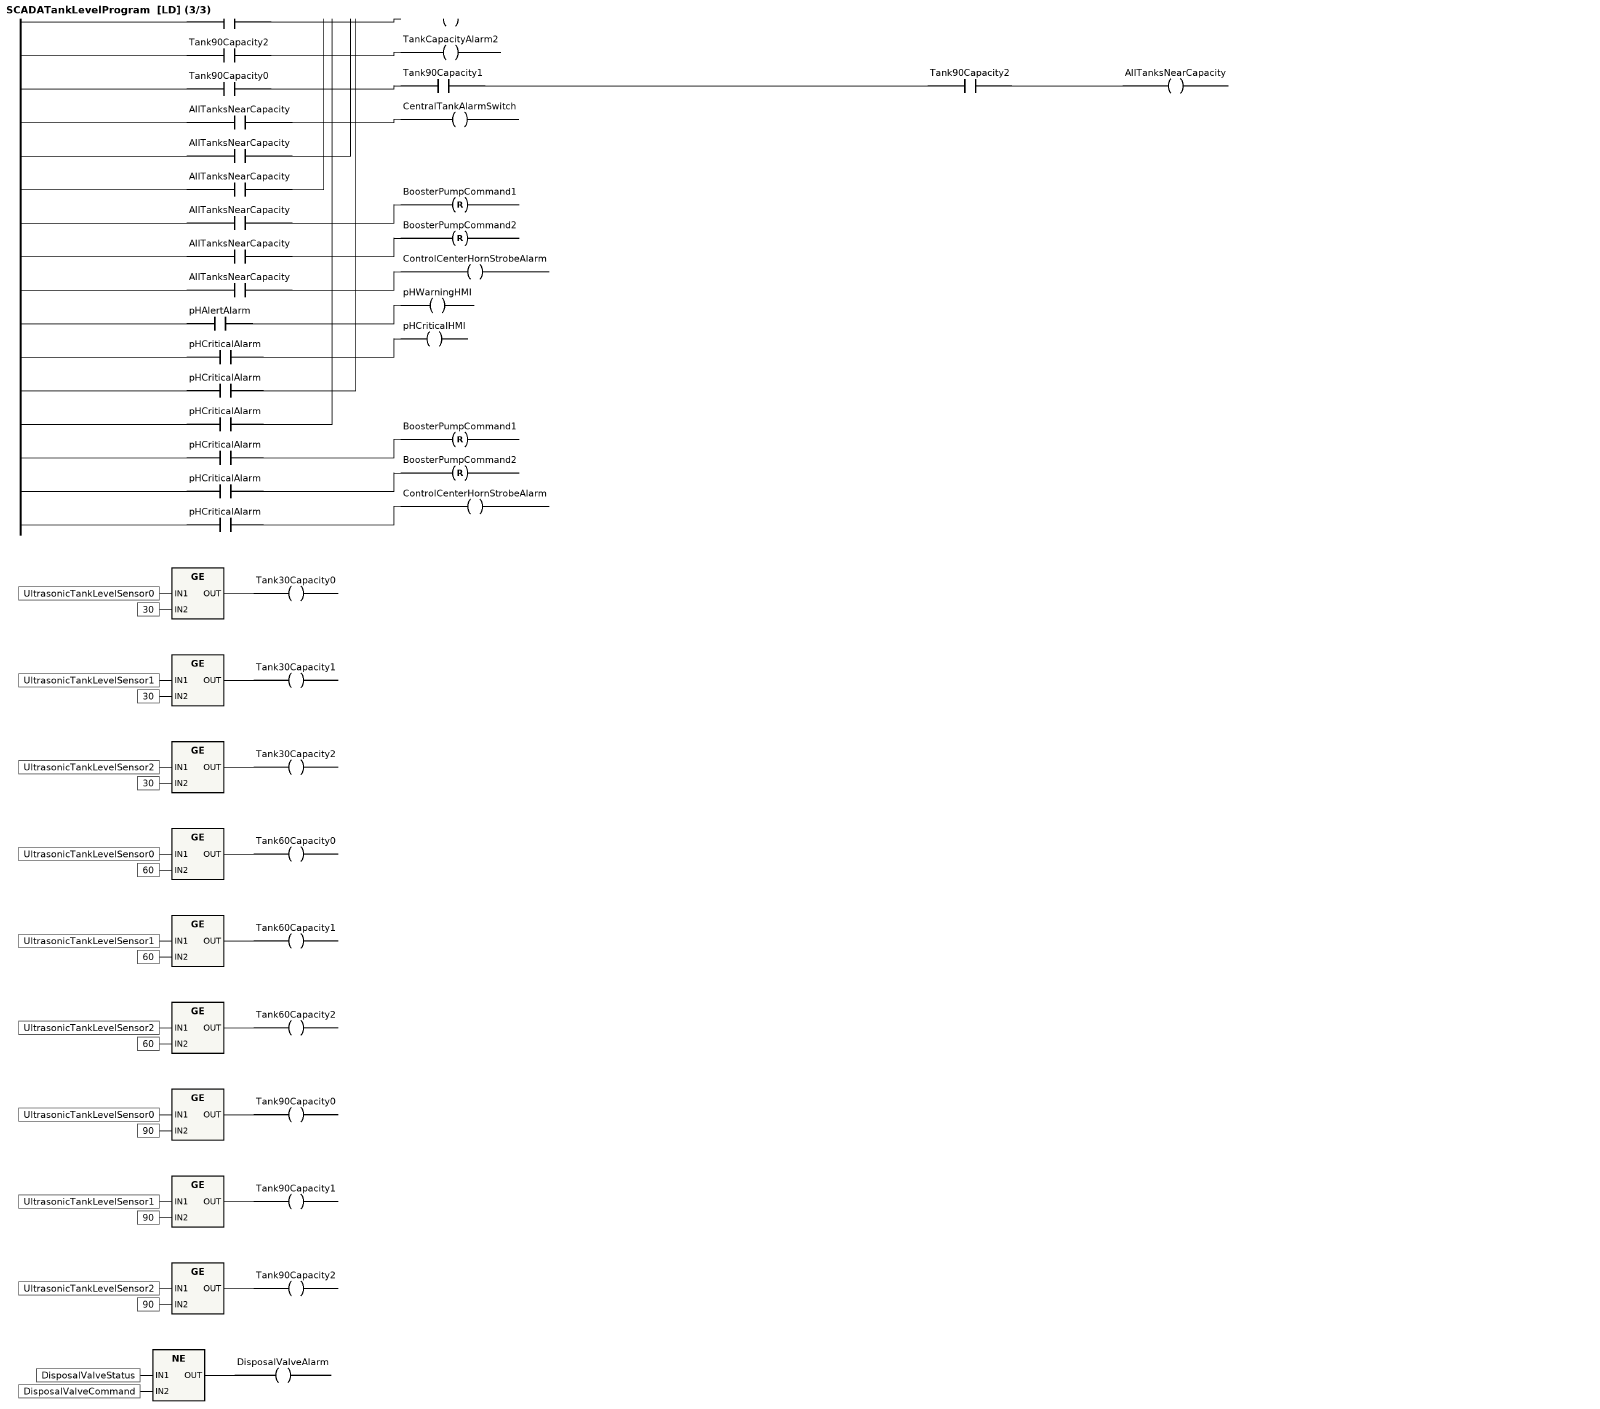
DisposalProtocol0(In := isContainmentUnitAttached, DistributionPumpSpeedIn := 50, DisposalValveCommandIn := 100);
DistributionPumpSpeedCommand := DisposalProtocol0.DistributionPumpSpeedOut;
_MOVE117_OUT := MOVE(EN := isTank1DisposalReady, IN := 0, ENO => _MOVE117_ENO);
IF _MOVE117_ENO THEN EductorValveCommand1 := _MOVE117_OUT; END_IF;
IF _MOVE117_ENO THEN DistributionPumpCommand := FALSE; END_IF;
_MOVE132_OUT := MOVE(EN := isTank2DisposalReady, IN := 0, ENO => _MOVE132_ENO);
IF _MOVE132_ENO THEN EductorValveCommand1 := _MOVE132_OUT; END_IF;
IF _MOVE132_ENO THEN DistributionPumpCommand := FALSE; END_IF;
isTank0DisposalReady := Tank30Capacity0 AND Tank60Capacity0 AND HMITankDisposalButton;
isTank1DisposalReady := Tank30Capacity1 AND Tank60Capacity1 AND HMITankDisposalButton;
isTank2DisposalReady := Tank30Capacity2 AND Tank60Capacity2 AND HMITankDisposalButton;
askHMIContainmentUnitAttached := isTank2DisposalReady OR isTank1DisposalReady OR isTank0DisposalReady;
DisposalValveCommand := DisposalProtocol0.DisposalValveCommandOut;
askHMIContainmentUnitFull := DisposalProtocol0.Out;
DisposalProtocol1(In := isContainmentUnitFull, DistributionPumpSpeedIn := 0, DisposalValveCommandIn := 0);
DisposalValveCommand := DisposalProtocol1.DisposalValveCommandOut;
DistributionPumpSpeedCommand := DisposalProtocol1.DistributionPumpSpeedOut;
DisposalValveAlarm := DisposalValveStatus <> DisposalValveCommand;
TankCapacityAlarm0 := Tank90Capacity0;
(* Checks to see if a tank has reached 90% capacity. If so, alarm for associated tank is set high and protocol is followed as if it were at a 60% (60) capacity. *)
TankCapacityAlarm1 := Tank90Capacity1;
TankCapacityAlarm2 := Tank90Capacity2;
(* Checks for the critical state of if all tanks are at 90% (90) capacity. This starts the emergency shutdown protocol which closes all valves and set all pumps to low, including the DCS valves and pumps utilzing global variables. This also engages associated alarms and horns for the critical condition. *)
AllTanksNearCapacity := Tank90Capacity0 AND Tank90Capacity1 AND Tank90Capacity2;
CentralTankAlarmSwitch := AllTanksNearCapacity;
_MOVE200_OUT := MOVE(EN := AllTanksNearCapacity, IN := 0, ENO => _MOVE200_ENO);
IF _MOVE200_ENO THEN EductorValveCommand0 := _MOVE200_OUT; END_IF;
EductorValveCommand1 := EductorValveCommand0;
EductorValveCommand2 := EductorValveCommand1;
IF _MOVE200_ENO THEN DistributionPumpCommand := FALSE; END_IF;
_MOVE111_OUT := MOVE(EN := AllTanksNearCapacity, IN := 0, ENO => _MOVE111_ENO);
IF _MOVE111_ENO THEN IsolationValveCommand0 := _MOVE111_OUT; END_IF;
IsolationValveCommand1 := IsolationValveCommand0;
IsolationValveCommand2 := IsolationValveCommand1;
IF _MOVE111_ENO THEN BoosterPumpCommand0 := FALSE; END_IF;
IF AllTanksNearCapacity THEN BoosterPumpCommand1 := FALSE; END_IF;
IF AllTanksNearCapacity THEN BoosterPumpCommand2 := FALSE; END_IF;
ControlCenterHornStrobeAlarm := AllTanksNearCapacity;
(* Utilizing the pH asynchronous program, this main program recieves alarm variables from that program and acts accordingly. The system pushes a warning to the HMI in the event of an alert. And a full system shutdown in the event of a critical pH alarm. *)
pHWarningHMI := pHAlertAlarm;
pHCriticalHMI := pHCriticalAlarm;
_MOVE143_OUT := MOVE(EN := pHCriticalAlarm, IN := 0, ENO => _MOVE143_ENO);
IF _MOVE143_ENO THEN DistributionPumpCommand := FALSE; END_IF;
_MOVE156_OUT := MOVE(EN := pHCriticalAlarm, IN := 0, ENO => _MOVE156_ENO);
IF _MOVE156_ENO THEN BoosterPumpCommand0 := FALSE; END_IF;
IF pHCriticalAlarm THEN BoosterPumpCommand1 := FALSE; END_IF;
IF pHCriticalAlarm THEN BoosterPumpCommand2 := FALSE; END_IF;
IF _MOVE143_ENO THEN EductorValveCommand0 := _MOVE143_OUT; END_IF;
EductorValveCommand1 := EductorValveCommand0;
EductorValveCommand2 := EductorValveCommand1;
IF _MOVE156_ENO THEN IsolationValveCommand0 := _MOVE156_OUT; END_IF;
IsolationValveCommand1 := IsolationValveCommand0;
IsolationValveCommand2 := IsolationValveCommand1;
ControlCenterHornStrobeAlarm := pHCriticalAlarm;
END_PROGRAM

FUNCTION isOutsidePHRange : BOOL
  VAR_INPUT
    EvalulateVarIn : INT;
    BasicMax : INT;
    AcidicMax : INT;
  END_VAR

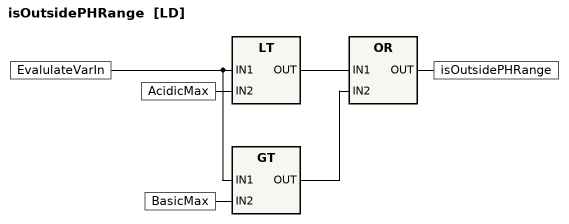
(* LD diagram, written out as Structured Text *)
isOutsidePHRange := EvalulateVarIn < AcidicMax OR EvalulateVarIn > BasicMax;
END_FUNCTION

PROGRAM SCADApHTankMonitorProgram
  VAR
    pHSensor AT %IW13 : INT := 7;
  END_VAR
  VAR CONSTANT
    AcidicLevel AT %MW3 : INT := 4;
    CriticalAcidicLevel AT %MW4 : INT := 3;
    BasicLevel AT %MW5 : INT := 10;
    CriticalBasicLevel AT %MW6 : INT := 11;
  END_VAR
  VAR_EXTERNAL
    pHAlertAlarm : BOOL;
    pHCriticalAlarm : BOOL;
  END_VAR

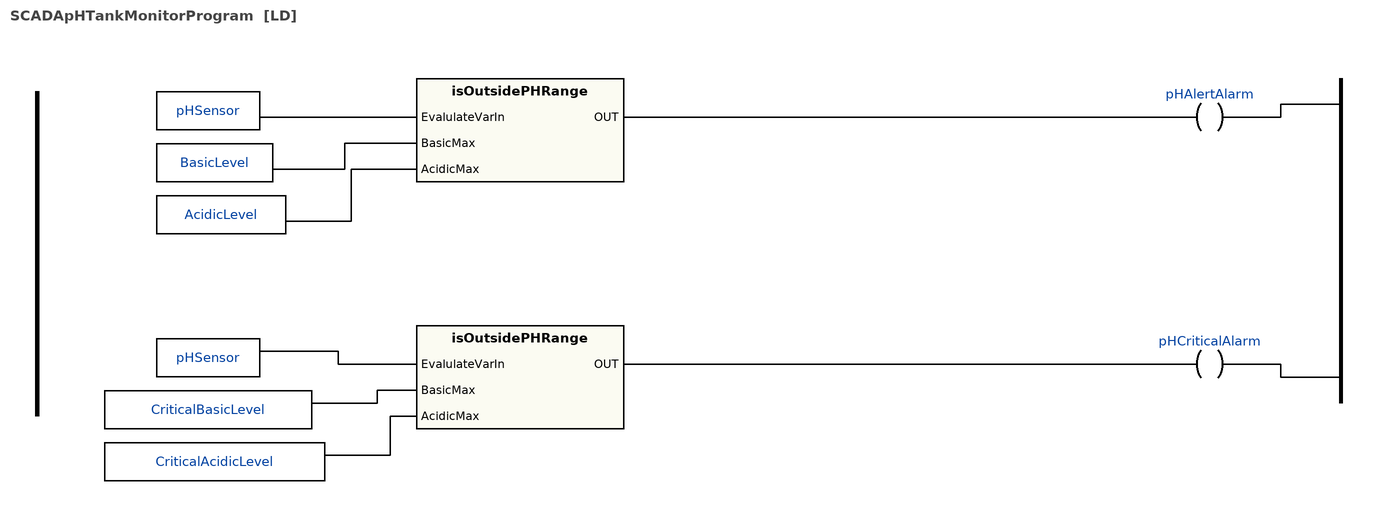
(* LD diagram, written out as Structured Text *)
pHAlertAlarm := isOutsidePHRange(pHSensor, BasicLevel, AcidicLevel);
pHCriticalAlarm := isOutsidePHRange(pHSensor, CriticalBasicLevel, CriticalAcidicLevel);
END_PROGRAM

CONFIGURATION Config0
  VAR_GLOBAL
    BoosterPumpCommand0 AT %QX0.0 : BOOL;
    BoosterPumpCommand1 AT %QX0.1 : BOOL;
    BoosterPumpCommand2 AT %QX0.2 : BOOL;
    IsolationValveCommand0 AT %QW10 : INT;
    IsolationValveCommand1 AT %QW11 : INT;
    IsolationValveCommand2 AT %QW12 : INT;
    pHAlertAlarm AT %QX0.3 : BOOL;
    pHCriticalAlarm AT %QX0.4 : BOOL;
  END_VAR
  RESOURCE Res0 ON PLC
    TASK task0(INTERVAL := T#20ms, PRIORITY := 0);
    TASK task1(INTERVAL := T#20ms, PRIORITY := 0);
    TASK task2(INTERVAL := T#20ms, PRIORITY := 0);
    PROGRAM instance0 WITH task0 : DCSProgramSector;
    PROGRAM instance1 WITH task1 : SCADATankLevelProgram;
    PROGRAM instance2 WITH task2 : SCADApHTankMonitorProgram;
  END_RESOURCE
END_CONFIGURATION
